FUNCTION_BLOCK SpeedSp (* Basic Function Block Type *)
  (* Standard: 61499-2 *)
  (* Version 0.0, 7/3/2026, Schneider Electric, Template *)
  PACKAGE SE.Nereda;
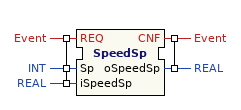
  EVENT_INPUT
    REQ WITH Sp, iSpeedSp; (* Normal Execution Request *)
  END_EVENT
  EVENT_OUTPUT
    CNF WITH oSpeedSp; (* Execution Confirmation *)
  END_EVENT
  VAR_INPUT
    Sp : INT;
    iSpeedSp : REAL;
  END_VAR
  VAR_OUTPUT
    oSpeedSp : REAL;
  END_VAR
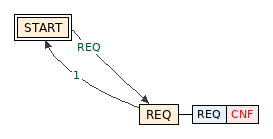
  EC_STATES
    START; (* Initial State *)
    REQ : REQ -> CNF; (* Normal execution *)
  END_STATES
  EC_TRANSITIONS
    START TO REQ := REQ;
    REQ TO START := 1;
  END_TRANSITIONS
  ALGORITHM INIT IN ST: (* Initialization algorithm *)
;
  END_ALGORITHM
  ALGORITHM REQ IN ST: (* Normally executed algorithm *)
;
IF Sp = 0 THEN
	oSpeedSp := 0;
ELSE
	oSpeedSp := iSpeedSp;
END_IF;
  END_ALGORITHM
END_FUNCTION_BLOCK
